FUNCTION_BLOCK SM_AxesIO
VAR_INPUT
	///Is control enabled?
	{attribute 'OPC.UA.DA' := '1'}
	{attribute 'OPC.UA.DA.Access' := '1'}
	isEnabled: BOOL;
END_VAR
VAR_OUTPUT
	///Current status description
	{attribute 'OPC.UA.DA' := '1'}
	{attribute 'OPC.UA.DA.Access' := '1'}
	actualStatus: STRING;
	///Statuses of the state machine
	statuses: AxesIOStatuses;
	///Parts of the state machine
	parts: AxesIOParts;
END_VAR
VAR_IN_OUT
END_VAR
VAR
END_VAR

parts.aziDrive( isEnabled := isEnabled );
parts.ablDrive( isEnabled := isEnabled );
parts.eleDrive( isEnabled := isEnabled );
statuses.healthStatus( isGood := parts.aziDrive.statuses.healthStatus.isGood AND (parts.ablDrive.statuses.healthStatus.isGood AND parts.eleDrive.statuses.healthStatus.isGood) );

END_FUNCTION_BLOCK

(* stored: Version 1.1.0.1, ProductVersion 3.1.4019.2
   POU SM_AxesIO: Id {ff125399-245d-4752-8b71-ab220430527b}, SpecialFunc None *)
